(*
	RJM Maszyny sp. z o.o.
	autor 	: Rafał Osajda
	data	: 02.02.2024
	TC		: 3.1 4024.54
	wersja	: 0.0.1.0	: pełna obsługa

	Obsługa elektrozaworu do sterowania siłownikiem pneumatycznym. FB bazowy dla pozostałych rodzajów elektrozaworów
*)
FUNCTION_BLOCK ABSTRACT FB_IOElectrovalve EXTENDS FB_BaseComponent IMPLEMENTS  ITF_IOElectrovalve, ITF_IOElectrovalve_HMI_Init
VAR
	bCoilA							AT %Q*	: BOOL;
	bCoilB							AT %Q*	: BOOL;
	eType									: E_IOElectrovalveType;
END_VAR

(*
	RJM Maszyny sp. z o.o.
	autor 	: Rafał Osajda
	data	: 21.02.2024
	TC		: 3.1 4024.54
	wersja	: 0.0.1.0	: pełna obsługa

	Ustawienie odpowiednich wyjść
*)
METHOD Contol : BOOL
VAR_INPUT
	eAction	: E_IOElectrovalveAction;
END_VAR
END_METHOD

METHOD PUBLIC GetElectrovalveType : E_IOElectrovalveType
VAR_INPUT
END_VAR
GetElectrovalveType			:= THIS^.eType;
END_METHOD

METHOD PUBLIC GetElectrovalveTypeToString : STRING
VAR CONSTANT
	arrType		: ARRAY [0..5] OF STRING := ['NC_3na2', 'NO_3na2', 'C1_5na2', 'C2_5na2', 'C2_5na3O', 'C2_5na3Z'];
END_VAR
GetElectrovalveTypeToString			:= arrType [TO_INT (THIS^.eType)];
END_METHOD

METHOD IsActiveCoilA : BOOL
VAR_INPUT
END_VAR
IsActiveCoilA			:= THIS^.bCoilA;
END_METHOD

METHOD IsActiveCoilB : BOOL
VAR_INPUT
END_VAR
IsActiveCoilB			:= THIS^.bCoilB;
END_METHOD

END_FUNCTION_BLOCK

(* stored: Version 1.1.0.1
   POU FB_IOElectrovalve: Id {ab7faff1-27f9-0552-30db-a3ee03923e14}, SpecialFunc None
   Folder ITF_Electrovalve_HMI_Connector: Id {a1d6ab22-3179-4649-9c0b-995a03a33f53}
   Method Contol: Id {05101fa4-1b68-0522-344f-bfe6ed566f1a}
   Method GetElectrovalveType: Id {014a69c7-7219-4234-8c0c-36b58219e3c9}
   Method GetElectrovalveTypeToString: Id {debc1117-cfe7-4a5c-b55c-0e8daa5df6ba}
   Method IsActiveCoilA: Id {15a459f2-566d-4208-ab88-8334c1bb7aa4}
   Method IsActiveCoilB: Id {7203c2d0-cd87-4264-b035-36bda2e9f593} *)
